Fanuc KAREL source: kt00263.KL

-- PROVISIONAL review KL for V770-1; original PC SHA256 b2dcc813c8432c705badb75aaed3b7b223b65ee1fb629659de03d90b1148e4d3
-- Incomplete behavior may be omitted. Consult companion uncertainty JSON. Do not deploy.
PROGRAM KT00263
%NOLOCKGROUP
VAR
  R1 : REAL
  OUT : BOOLEAN
-- UNRESOLVED_DECL Y2 type=002018
BEGIN
  -- UNRESOLVED_PC offsets 5-16; opcodes 2E,23
  -- UNRESOLVED_PC offsets 21-35; opcodes 2E,22,9D,33,B2
  -- UNRESOLVED_PC offsets 40-63; opcodes 21,22,9D,33,B1,64,6D,23
  -- UNRESOLVED_PC offsets 68-72; opcodes 7F
END KT00263
